(* CODESYS project youtube_alexa_stepper_example.ecp

Project tree, tasks and I/O mapping:
  PFC100_2ETH_RS : 750-8102 PFC100 CS 2ETH RS, WAGO, order no. 0750-8102, version 5.11.1.16
    application Application
      libraries: ; WagoAppStepper, * (WAGO); WagoAppCloud, 1.2.4.13 (WAGO); WagoSysPlainMem, * (WAGO); WagoSysString, * (WAGO)
      task PLC_Task (cyclic, interval t#50ms, priority 15) calls PLC_PRG
      program PLC_PRG [ST]
      program STEPPER_PRG [ST]
      program MQTT_PRG [ST]
      function block UPDATE_AWS_IOT_THING_SHADOW [ST]: PUB_STRING
      data type typIOT_THING_SHADOW
      global variables GVL
    DeviceAdapter
    Kbus : Kbus, WAGO, version 1.4.0.2
        unmapped channels: K-BUS diagnostics
      Servo_Stepper_Controller_55_VDC_7_5A : 0750-0673, WAGO, order no. 0750-0673, version 0.0.0.19
          settings: K-BUS Module slot index = 1
          unmapped channels: status byte S0, speed, process value, status byte S3, status byte S2, status byte S1, control byte C0, speed, acceleration, process value, control byte C3, control byte C2, control byte C1
        DeviceAdapter
    MODBUS
      MODBUS : MODBUS, WAGO, order no. n/a, version 1.1.1.15
    Serial
      COM1 : COM1, WAGO, version 0.0.0.19
*)

// PFC100_2ETH_RS/Application/typIOT_THING_SHADOW
TYPE typIOT_THING_SHADOW :
STRUCT
		sLabel	: STRING;
		sValue	: STRING;
END_STRUCT
END_TYPE

// PFC100_2ETH_RS/Application/GVL
{attribute 'qualified_only'}
VAR_GLOBAL
	Shadow_Attributes	: ARRAY[1..20] OF typIOT_THING_SHADOW;
	rtNewMqttData		: R_TRIG;
END_VAR

// PFC100_2ETH_RS/Application/PLC_PRG
PROGRAM PLC_PRG
VAR
END_VAR

STEPPER_PRG();
MQTT_PRG();

END_PROGRAM

// PFC100_2ETH_RS/Application/STEPPER_PRG
PROGRAM STEPPER_PRG
VAR
	//stepper variables
	fbStepperControl		: WagoAppStepper.FbStepperControlBasic;
	xStepperEnable			: BOOL;
	eStepperMode			: eMode 	:= eMode.MoveAbsolute;
	xStepperDirectionPos	: BOOL		:= TRUE;
	xStepperDirectionNeg	: BOOL		:= FALSE;
	iStepperSpeedCmd		: INT		:= 25000;
	wStepperAccelCmd		: WORD 		:= 15000;
	wStepperDecelCmd		: WORD 		:= 15000;
	diStepperPositionCmd	: DINT;
	xStepperRunTrig			: BOOL;
	xStepperErrorResetTrig	: BOOL;
	xStepperStopCmd			: BOOL;
	xStepperIsFinished		: BOOL;
	xStepperIsBusy			: BOOL;
	xStepperIsError			: BOOL;
	oStepperStatus			: WagoSysErrorBase.FbResult;
	//eStepperErrorCode		: eStatus;
	diStepperActualPosition	: DINT;
	iStepperActualSpeed		: INT;
	xStepperMbIsActive		: BOOL;
	xStepperResetWarning	: BOOL;
	//eStepperErrorCode		: eStatus;
	diStepperPositionCmdOld: DINT;
	rtStepperInPosition: R_TRIG;
END_VAR

fbStepperControl(
	xEnable:= xStepperEnable, 
	I_Port:= IoConfig_Globals.Servo_Stepper_Controller_55_VDC_7_5A, 
	eJobType:= eStepperMode, 
	xDirPos:= xStepperDirectionPos, 
	xDirNeg:= xStepperDirectionNeg, 
	iSpeed:= iStepperSpeedCmd, 
	wAcceleration:= wStepperAccelCmd, 
	wDeceleration:= wStepperDecelCmd, 
	diPosition:= diStepperPositionCmd, 
	xTriggerStart:= xStepperRunTrig, 
	xTriggerErrorReset:= xStepperErrorResetTrig, 
	xStop:= xStepperStopCmd, 
	xJobFinished=> xStepperIsFinished, 
	xBusy=> xStepperIsBusy, 
	xError=> xStepperIsError, 
	oStatus=> oStepperStatus, 
	eErrorCodes=> , 
	diActualPosition=> diStepperActualPosition, 
	iActualSpeed=> iStepperActualSpeed, 
	xMailboxActive=> xStepperMbIsActive, 
	xResetWarning=> xStepperResetWarning);
	
	diStepperPositionCmd := STRING_TO_DINT(GVL.Shadow_Attributes[2].sValue);
	
	IF diStepperPositionCmd <> diStepperPositionCmdOld THEN
		xStepperEnable := TRUE;
		xStepperRunTrig := TRUE;
	END_IF
	
	rtStepperInPosition(CLK:= xStepperIsFinished);
	IF rtStepperInPosition.Q THEN
		xStepperEnable := FALSE;
		diStepperPositionCmdOld := diStepperPositionCmd;
	END_IF

END_PROGRAM

// PFC100_2ETH_RS/Application/MQTT_PRG
PROGRAM MQTT_PRG
VAR
	fbMQTT_Sub						: WagoAppCloud.FbSubscribeMQTT;
	
	sMqttSubTopic					: STRING(255) := '$$aws/things/WAGO_ALEXA/shadow/update/accepted';
	
	eMqttSubQoS: eQualityOfService 	:= 0;
	aMqttSubPayloadData				: ARRAY[0..1000] OF BYTE;
	xMqttSubIsBusy					: BOOL;
	xMqttSubIsSubscribed			: BOOL;
	xMqttSubError					: BOOL;
	oMqttSubStatus					: WagoSysErrorBase.FbResult;
	xMqttSubIsData					: BOOL;
	dwMqttSubRcvSize				: DWORD;
	xMqttSubDataTruncated			: BOOL;
	xMqttSubEnable					: BOOL;

//*********************************************
	xConvertToTyp: BOOL;
	b: UDINT;
	xByteIsChar: BOOL;
	iCurlIndex: INT;
	xOnLabel: BOOL;
	xOnValue: BOOL;
	iWriteIndex: INT;
	sCurrentValueString: STRING;
	sCurrentLabelString: STRING;
	ub: DINT;
	rtNewData			: R_TRIG;
	sMqttSubRcvString	: STRING(255);
END_VAR

fbMQTT_Sub(
	xSubscribe:= xMqttSubEnable, 
	sTopic:= sMqttSubTopic, 
	eQoS:= eMqttSubQoS, 
	aPayloadData:= aMqttSubPayloadData, 
	xBusy=> xMqttSubIsBusy, 
	xIsSubscribed=> xMqttSubIsSubscribed, 
	xError=> xMqttSubError, 
	oStatus=> oMqttSubStatus, 
	xDataReceived=> xMqttSubIsData, 
	dwRxNBytes=> dwMqttSubRcvSize, 
	xDataTruncated=> xMqttSubDataTruncated);
	
	xMqttSubEnable := TRUE;
	
	GVL.rtNewMqttData(CLK:= xMqttSubIsData);
	
	IF GVL.rtNewMqttData.Q THEN
		// copy the ASCII data to a string
		MemCopy(ADR(sMqttSubRcvString), ADR(aMqttSubPayloadData),dwMqttSubRcvSize);
	
		FOR b := 0 TO DWORD_TO_INT(dwMqttSubRcvSize) DO
			//checks to see if the byte is an alpha-numeric
			IF 	((aMqttSubPayloadData[b] >= 48) AND aMqttSubPayloadData[b] <= 57) 	OR
				((aMqttSubPayloadData[b] >= 65) AND aMqttSubPayloadData[b] <= 90) 	OR
				((aMqttSubPayloadData[b] >= 97) AND aMqttSubPayloadData[b] <= 122) 	THEN
				xByteIsChar := TRUE;
			ELSE
				xByteIsChar := FALSE;
			END_IF
					
		// curly braces
			IF (aMqttSubPayloadData[b] = 123) THEN
				iCurlIndex := iCurlIndex + 1;
			END_IF
			
			// if this is a new scan or the byte is a comma
			IF ((iCurlIndex = 3) AND ((aMqttSubPayloadData[b] = 123))  OR (aMqttSubPayloadData[b] = 44) AND NOT xOnLabel) THEN
				xOnLabel := TRUE;
				xOnValue := FALSE;
				GVL.Shadow_Attributes[iWriteIndex].sLabel:= sCurrentLabelString;
				GVL.Shadow_Attributes[iWriteIndex].sValue:= sCurrentValueString;
				sCurrentLabelString := '';
				sCurrentValueString := '';
				iWriteIndex := iWriteIndex + 1;
					
			//looks for a colon
			ELSIF (aMqttSubPayloadData[b] = 58) THEN
				xOnLabel := FALSE;
				xOnValue := TRUE;
			END_IF
					
			IF xByteIsChar THEN
				IF xOnLabel THEN
					sCurrentLabelString := CONCAT(sCurrentLabelString, ASCIIBYTE_TO_STRING(aMqttSubPayloadData[b]));
				ELSIF xOnValue THEN
					sCurrentValueString := CONCAT(sCurrentValueString, ASCIIBYTE_TO_STRING(aMqttSubPayloadData[b]));
				END_IF
			END_IF
	
			IF iWriteIndex > 2 THEN
				xOnLabel := FALSE;
				xOnValue := FALSE;
				iCurlIndex := 0;
				iWriteIndex := 0;
				RETURN;
			END_IF
		END_FOR
	END_IF

END_PROGRAM

// PFC100_2ETH_RS/Application/UPDATE_AWS_IOT_THING_SHADOW
FUNCTION_BLOCK UPDATE_AWS_IOT_THING_SHADOW
VAR_IN_OUT
	xExecute: BOOL;	// trigger to send the data to the AWS IoT Thing Shadow
	Shadow_Attributes	: ARRAY[*] OF typIOT_THING_SHADOW;
END_VAR
VAR_INPUT
	sRootCaPath			: STRING;
	sCertPath			: STRING;
	sKeyPath			: STRING;
	sEndpoint			: STRING;
	sTopic				: STRING;
END_VAR
VAR
	fbWriteFile			: FbWriteWholeFile_cpt;
	ub					: DINT;
	lb					: DINT;
	i					: DINT;
	sBaseString			: STRING(22) := '{"state":{"reported":{ ';
	sAttributeString	: STRING;
	aWriteBytes			: ARRAY[1..10000] OF BYTE;
	aHoldBytes			: ARRAY[1..80] OF BYTE;
	ptString 			: POINTER TO BYTE;
	l					: INT;
	diSizeOfString		: DINT;
	index				: INT;
	x: INT;
	sTestString: STRING(255);
	xWriteFile: BOOL;
	oWriteFileStatus: FbResult;
	xWriteFileTrig: BOOL;
	xWriteFileError: BOOL;
	xWriteFileBusy: BOOL;
	sWriteFileName: STRING := '/root/.send_shadow.json';
	sPublishBashScript: STRING(255);
	rtsSendResult: RTS_IEC_RESULT;
	sReturnResponse: STRING(255);
END_VAR

ub:=UPPER_BOUND (Shadow_Attributes,1);
lb:=LOWER_BOUND (Shadow_Attributes,1);

IF xExecute THEN
	index := 0;
	//begin building the array
	ptString := ADR(sBaseString);
	FOR l := 1 TO len(sBaseString) DO
		aWriteBytes[l] := ptString^;
		ptString := ptString + 1;
	END_FOR	
	ptString := 0;
	index := index + len(sBaseString);
	// write JSON header
	FOR i := lb TO ub DO /// loop through each atrribute / value
		sAttributeString := '"';
		sAttributeString := CONCAT(sAttributeString, Shadow_Attributes[i].sLabel);
		sAttributeString := CONCAT(sAttributeString, '": "');
		sAttributeString := CONCAT(sAttributeString, Shadow_Attributes[i].sValue);
		sAttributeString := CONCAT(sAttributeString, '"');
		IF (i < ub) THEN
			sAttributeString := CONCAT(sAttributeString, ',');
		ELSIF i = ub THEN
			sAttributeString := CONCAT(sAttributeString, '}}}');
		END_IF
		diSizeOfString := LEN(sAttributeString);
		ptString := ADR(sAttributeString);
		FOR l := 1 TO len(sAttributeString) DO
			aHoldBytes[l] := ptString^;
			ptString := ptString + 1;
			aWriteBytes[l + index] := aHoldBytes[l]; 
		END_FOR
		
		index := index + len(sAttributeString);
		
		IF i = ub THEN
			xWriteFileTrig := TRUE;
		END_IF
	END_FOR

// write the file
	fbWriteFile(
		oStatus=> oWriteFileStatus, 
		xTrigger:= xWriteFileTrig, 
		xError=> xWriteFileError, 
		xBusy=> xWriteFileBusy, 
		sName:= sWriteFileName, 
		pTxBuffer:= ADR(aWriteBytes), 
		udiTxNBytes:= index);
		
		IF NOT xWriteFileTrig THEN
			sPublishBashScript := PUB_STRING(
										sRootCaPath:= sRootCaPath, 
										sCertPath:= sCertPath, 
										sKeyPath:= sKeyPath, 
										sEndPoint:= sEndpoint, 
										sTopic:= sTopic);
			SysProcessExecuteCommand2(pszCommand:= sPublishBashScript, pszStdOut:= sReturnResponse, udiStdOutLen:= 255, pResult:= rtsSendResult);
			xExecute := FALSE;
		END_IF
END_IF

METHOD INTERNAL PUB_STRING : STRING(255)
VAR_INPUT
	sRootCaPath	: STRING;
	sCertPath	: STRING;
	sKeyPath	: STRING;
	sEndPoint	: STRING;
	sTopic		: STRING;
END_VAR

VAR
	sHoldString: STRING(255);
END_VAR
//mosquitto_pub --cafile $1 --cert $2 --key $3 -h $4 -p 8883 -q 1 -d -t $5 -f $6
sHoldString := 'sh /root/.send_shadow.sh ';
sHoldString := CONCAT(sHoldString, sRootCaPath);
sHoldString := CONCAT(sHoldString, ' ');
sHoldString := CONCAT(sHoldString, sCertPath);
sHoldString := CONCAT(sHoldString, ' ');
sHoldString := CONCAT(sHoldString, sKeyPath);
sHoldString := CONCAT(sHoldString, ' ');
sHoldString := CONCAT(sHoldString, sEndPoint);
sHoldString := CONCAT(sHoldString, ' $'');
sHoldString := CONCAT(sHoldString, sTopic);
sHoldString := CONCAT(sHoldString, '$' /root/.send_shadow.json');

PUB_STRING := sHoldString;
END_METHOD

END_FUNCTION_BLOCK
